// TIA Portal V16 export
// export: Created 2022-02-04T14:40:09.0663123Z, ExportSetting WithDefaults, DisplayName Totally Integrated Automation Portal, DisplayVersion V16 Update 1, DisplayName TIA Portal Version Control Interface, DisplayVersion V16, DisplayName TIA Portal Openness, DisplayVersion V16, DisplayName SINAMICS Startdrive Advanced, DisplayVersion V16 Update 5, DisplayName SINAMICS Startdrive G130, G150, S120, S150, SINAMICS MV, S210, DisplayVersion V16 Update 5, DisplayName SINAMICS Startdrive G110M, G120, G120C, G120D, G120P, G115D, DisplayVersion V16 Update 5, DisplayName STEP 7 Professional, DisplayVersion V16, DisplayName STEP 7 Safety, DisplayVersion V16, DisplayName WinCC Advanced, DisplayVersion V16, DisplayName SIMATIC Visualization Architect, DisplayVersion V16
ORGANIZATION_BLOCK "PS_FLT"   // OB81, LAD, PowerSupplyError
TITLE = "Power Supply Fault"
VERSION : 0.1
// stored: IsIECCheckEnabled false
   VAR_TEMP
      OB81_EV_CLASS : Byte;   // 16#39, Event class 3, Entering event state, Internal fault event
      OB81_FLT_ID : Byte;   // 16#XX, Fault identifcation code
      OB81_PRIORITY : Byte;   // Priority of OB Execution
      OB81_OB_NUMBR : Byte;   // 81 (Organization block 81, OB81)
      OB81_RESERVED_1 : Byte;   // Reserved for system
      OB81_RESERVED_2 : Byte;   // Reserved for system
      OB81_RACK_CPU : Word;   // Bits 0 to 2: Rack no; Bit 3: 0=standby CPU, 1=master CPU; Bits 4 to 7: 1111
      OB81_RESERVED_3 : Byte;   // Reserved for system
      OB81_RESERVED_4 : Byte;   // Reserved for system
      OB81_RESERVED_5 : Byte;   // Reserved for system
      OB81_RESERVED_6 : Byte;   // Reserved for system
      OB81_DATE_TIME : Date_And_Time;   // Date and time OB81 started
   END_VAR
BEGIN
END_ORGANIZATION_BLOCK
